PROGRAM MAIN
VAR
    TestSuite : T_TestSuite;
END_VAR

TestSuite();

END_PROGRAM

(* stored: Version 1.1.0.1, ProductVersion 3.1.4024.12
   POU MAIN: Id {63470fcc-b57d-026d-334d-1963f895812d}, SpecialFunc None *)
